TYPE ST_JXE1_MovementFeedback :
STRUCT
	CurrentPosition		: T_JXCE1_Position;
	CurrentSpeed		: T_JXCE1_Position;
	CurrentPushingForce	: T_JXCE1_Force;
	TargetPosition		: T_JXCE1_Position;
END_STRUCT
END_TYPE

(* stored: Version 1.1.0.1, ProductVersion 3.1.4024.15
   DUT ST_JXE1_MovementFeedback: Id {a44bfa8c-4b7d-0d17-0750-2e95ece020be} *)
